{attribute 'GeneratedUsingTerminal: EL7041-1000-0021'}
{attribute addProperty BoxType "EL7041-1000-0021"}
{attribute addProperty Id "StatusAT %I*Status_8CBE219F12Counter_valueAT %I*UINT2Latch_valueAT %I*UINT2"}
{attribute addProperty CRC "1292267034"}
{attribute addProperty Size "16"}
TYPE ENC_Status_compact_4D066E1A EXTENDS TcoIo.InputBase_8311D824 :
STRUCT
	{attribute addProperty Name "Status"}
	Status AT %I* : Status_8CBE219F;
	{attribute addProperty Name "Counter_value"}
	Counter_value AT %I* : UINT;
	{attribute addProperty Name "Latch_value"}
	Latch_value AT %I* : UINT;
END_STRUCT
END_TYPE

(* stored: Version 1.2.0.0, ProductVersion 3.1.4024.11
   DUT ENC_Status_compact_4D066E1A: Id {76e1dd1d-bcae-0f44-26b6-d5a2cb654a8f} *)
